# EPICS substitutions: ecmcApp/Db/ecmcGeneral.substitutions
file "ecmcGeneral.template"
{
pattern
{P,      PORT}
{IOC2:,  MC_CPU1}
}
